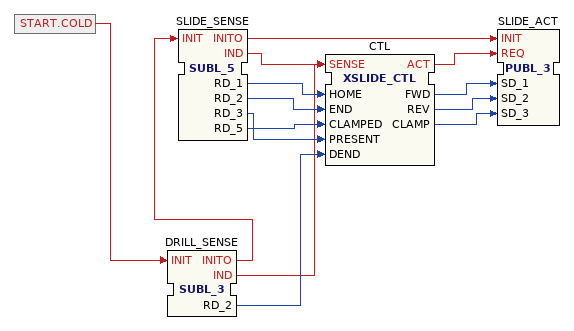
      [picture p28: resource CONTROL.SLIDE]
      FBS
        DRILL_SENSE : SUBL_3;
        SLIDE_SENSE : SUBL_5;
        CTL : XSLIDE_CTL;
        SLIDE_ACT : PUBL_3;
      END_FBS
      EVENT_CONNECTIONS
        START.COLD TO DRILL_SENSE.INIT;
        DRILL_SENSE.INITO TO SLIDE_SENSE.INIT;
        SLIDE_SENSE.INITO TO SLIDE_ACT.INIT;
        SLIDE_SENSE.IND TO CTL.SENSE;
        DRILL_SENSE.IND TO CTL.SENSE;
        CTL.ACT TO SLIDE_ACT.REQ;
      END_CONNECTIONS
      DATA_CONNECTIONS
        SLIDE_SENSE.RD_1 TO CTL.HOME;
        SLIDE_SENSE.RD_2 TO CTL.END;
        DRILL_SENSE.RD_2 TO CTL.DEND;
        CTL.FWD TO SLIDE_ACT.SD_1;
        CTL.REV TO SLIDE_ACT.SD_2;
        CTL.CLAMP TO SLIDE_ACT.SD_3;
        SLIDE_SENSE.RD_3 TO CTL.PRESENT;
        SLIDE_SENSE.RD_5 TO CTL.CLAMPED;
      END_CONNECTIONS
    END_RESOURCE
    RESOURCE DRILL : EMB_RES
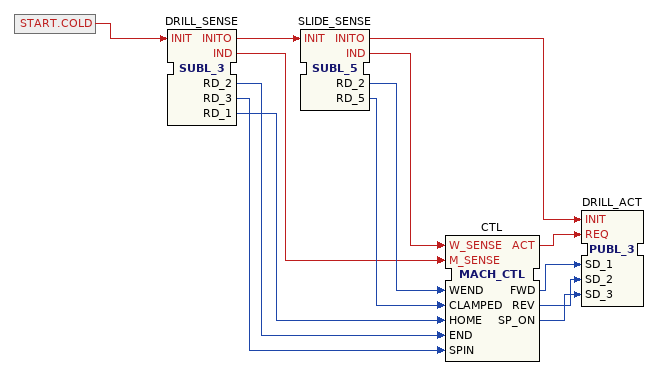
      FBS
        DRILL_SENSE : SUBL_3;
        SLIDE_SENSE : SUBL_5;
        CTL : MACH_CTL;
        DRILL_ACT : PUBL_3;
      END_FBS
      EVENT_CONNECTIONS
        START.COLD TO DRILL_SENSE.INIT;
        DRILL_SENSE.INITO TO SLIDE_SENSE.INIT;
        SLIDE_SENSE.INITO TO DRILL_ACT.INIT;
        SLIDE_SENSE.IND TO CTL.W_SENSE;
        DRILL_SENSE.IND TO CTL.M_SENSE;
        CTL.ACT TO DRILL_ACT.REQ;
      END_CONNECTIONS
      DATA_CONNECTIONS
        SLIDE_SENSE.RD_2 TO CTL.WEND;
        DRILL_SENSE.RD_2 TO CTL.END;
        DRILL_SENSE.RD_3 TO CTL.SPIN;
        CTL.FWD TO DRILL_ACT.SD_1;
        CTL.REV TO DRILL_ACT.SD_2;
        CTL.SP_ON TO DRILL_ACT.SD_3;
        SLIDE_SENSE.RD_5 TO CTL.CLAMPED;
        DRILL_SENSE.RD_1 TO CTL.HOME;
      END_CONNECTIONS
    END_RESOURCE
    RESOURCE UNLOAD : EMB_RES
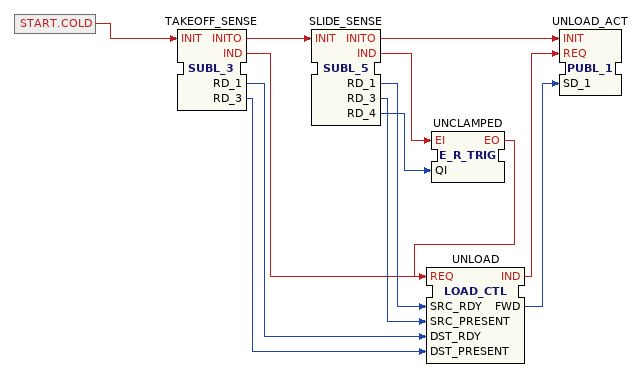
      FBS
        SLIDE_SENSE : SUBL_5;
        TAKEOFF_SENSE : SUBL_3;
        UNLOAD : LOAD_CTL;
        UNLOAD_ACT : PUBL_1;
        UNCLAMPED : E_R_TRIG;
      END_FBS
      EVENT_CONNECTIONS
        START.COLD TO TAKEOFF_SENSE.INIT;
        TAKEOFF_SENSE.INITO TO SLIDE_SENSE.INIT;
        SLIDE_SENSE.INITO TO UNLOAD_ACT.INIT;
        TAKEOFF_SENSE.IND TO UNLOAD.REQ;
        UNLOAD.IND TO UNLOAD_ACT.REQ;
        SLIDE_SENSE.IND TO UNCLAMPED.EI;
        UNCLAMPED.EO TO UNLOAD.REQ;
      END_CONNECTIONS
      DATA_CONNECTIONS
        TAKEOFF_SENSE.RD_1 TO UNLOAD.DST_RDY;
        TAKEOFF_SENSE.RD_3 TO UNLOAD.DST_PRESENT;
        SLIDE_SENSE.RD_1 TO UNLOAD.SRC_RDY;
        UNLOAD.FWD TO UNLOAD_ACT.SD_1;
        SLIDE_SENSE.RD_3 TO UNLOAD.SRC_PRESENT;
        SLIDE_SENSE.RD_4 TO UNCLAMPED.QI;
      END_CONNECTIONS
    END_RESOURCE
    RESOURCE TAKEOFF : EMB_RES
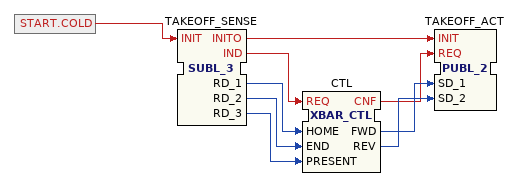
      FBS
        TAKEOFF_SENSE : SUBL_3;
        CTL : XBAR_CTL;
        TAKEOFF_ACT : PUBL_2;
      END_FBS
      EVENT_CONNECTIONS
        START.COLD TO TAKEOFF_SENSE.INIT;
        TAKEOFF_SENSE.INITO TO TAKEOFF_ACT.INIT;
        TAKEOFF_SENSE.IND TO CTL.REQ;
        CTL.CNF TO TAKEOFF_ACT.REQ;
      END_CONNECTIONS
      DATA_CONNECTIONS
        TAKEOFF_SENSE.RD_1 TO CTL.HOME;
        TAKEOFF_SENSE.RD_2 TO CTL.END;
        TAKEOFF_SENSE.RD_3 TO CTL.PRESENT;
        CTL.FWD TO TAKEOFF_ACT.SD_1;
        CTL.REV TO TAKEOFF_ACT.SD_2;
      END_CONNECTIONS
    END_RESOURCE
  END_DEVICE
END_SYSTEM
